TYPE TcaPushButtonStatus :
STRUCT
	LightState : eTcaPushButtonLightState;
	Light : BOOL;	
	Signal : BOOL;
	Raising : BOOL;
	Falling : BOOL;
	ElapsedTime : TIME;
END_STRUCT
END_TYPE

(* stored: Version 1.1.0.1
   DUT TcaPushButtonStatus: Id {990d3dc7-299a-4e6f-bf01-94b1ca04be70} *)
